TYPE ST_SG_Outputs_ProBOX :
(**************************************************************************************
 * 	Application		:	BoxControl Framework
 *	Revision		:	$Revision: $
 *	Revision date	:	$Date: $
 *	Last changed by	:	$Author: $
 *	URL				:	$URL: $
 *
 *	Purpose			:	Switching group - Outputs
 *
 * ------------------------------------------------------------------------------------
 *	Copyright Swisslog [IP AG], Switzerland. All rights reserved.
 * 
 * ------------------------------------------------------------------------------------
 *	
 * 	Revision History: 
 *
 * 	VERSION			DATE			INITIALS			DESCRIPTION
 *	0.1				01.01.2001		swl					Example
 *
 **************************************************************************************)
STRUCT
	GroupIsStarting			: BOOL;	// Group is starting (Can be used for warnings) 
	GroupStarted			: BOOL; // Group is starting or already started
	GroupStopped			: BOOL;	// Group is stopping or already stopped
	ErrorPending			: BOOL;	// Group or a member has an error 
	ResetPulse				: BOOL; // Reset pulse
	EmgStopStatus			: BOOL;	// Emergency lamp status
END_STRUCT
END_TYPE

(* stored: Version 1.1.0.1, ProductVersion 3.1.4024.9
   DUT ST_SG_Outputs_ProBOX: Id {2df61800-57bb-480f-b879-18a216e1a698} *)
